// Implicitly generated code : DO NOT EDIT
FUNCTION CheckRangeUnsigned : UDINT
VAR_INPUT
	value, lower, upper: UDINT;
END_VAR

// Implicitly generated code : Only an Implementation suggestion
{noflow}
IF (value < lower) THEN
	CheckRangeUnsigned := lower;
ELSIF(value > upper) THEN
	CheckRangeUnsigned := upper;
ELSE
	CheckRangeUnsigned := value;
END_IF
{flow}

END_FUNCTION

(* stored: Version 1.1.0.1, ProductVersion 3.1.4024.11
   POU CheckRangeUnsigned: Id {c54c921e-2f76-4e75-89d0-07a5dc8f40f2}, SpecialFunc CheckRangeUnsigned *)
